PROGRAM MAIN
VAR
	stTank1 : ST_Tank := (nId := 101,fTemperature := 80.3, fLevel := 80, bAlarm := FALSE );
	stTank2 : ST_Tank  := (nId := 102,fTemperature := 72.5, fLevel := 70, bAlarm := FALSE );
	stTank3 : ST_Tank  := (nId := 103,fTemperature := 90.8, fLevel := 90, bAlarm := FALSE );
	
	fbController1 : FB_TankController(stTank1);
	fbController2 : FB_TankController(stTank2);
	fbController3 : FB_PressureTankController(stTank3);
	
	aTankArray : ARRAY[1..cNUMBER_OF_TANKS] OF I_TankController := [fbController1, fbController2, fbController3];
	i : INT ;
	bStart : bool;
END_VAR
VAR CONSTANT
	cNUMBER_OF_TANKS :INT :=3;
END_VAR

IF bStart THEN
	FOR i := 1 TO cNUMBER_OF_TANKS DO
		IF aTankArray[i] <> 0 THEN
			aTankArray[i].StartController();
		END_IF
	END_FOR
	bStart := FALSE;
END_IF

END_PROGRAM

(* stored: Version 1.1.0.1, ProductVersion 3.1.4024.16
   POU MAIN: Id {2c746bd3-19f4-4202-bd9b-780eacf3677c}, SpecialFunc None *)
